{attribute 'qualified_only'}
{attribute 'strict'}
TYPE E_MixingValveControlMode :
(
	position := 0,
	heating := 1,
	cooling := 2
);
END_TYPE

(* stored: Version 1.1.0.1, ProductVersion 3.1.4024.9
   DUT E_MixingValveControlMode: Id {463072c4-69fe-4cca-86b0-8e2f9e26a76b} *)
